Fanuc KAREL source: kt00550.KL

-- PROVISIONAL review KL for V770-1; original PC SHA256 4c93fdad7d8666b9835c9394ab7483b163634d4435c1b10920c9b006a73b3c12
-- Incomplete behavior may be omitted. Consult companion uncertainty JSON. Do not deploy.
PROGRAM KT00550
%NOLOCKGROUP
-- UNRESOLVED_DECL P1 type=000199
-- UNRESOLVED_DECL P2 type=000199
-- UNRESOLVED_DECL OUT type=000102
BEGIN
  -- UNRESOLVED_PC offsets 5-44; opcodes 49,7E,49,7E,60,7E,4A
  -- UNRESOLVED_PC offsets 49-53; opcodes 7F
END KT00550
